Universal Robots PolyScope program: target_pose_tracking.urp

Program target_pose_tracking (createdIn=3.5.4.10845 lastSavedIn=3.5.4.10845 directory=/home/ur/ursim-current/programs installation=default robotSerialNumber=2014309999)
Calibrated DH parameters: a=[0, -0.612, -0.5723, 0, 0, 0]; d=[0.1273, 0, 0, 0.163941, 0.1157, 0.0922]; alpha=[1.570796, 0, 0, 1.570796, -1.570796, 0]; deltaTheta=[0, 0, 0, 0, 0, 0]
BeforeStart
  target_pose := Joint_6_name
  Popup Message (haltProgram=false message=Program has started from the beginning :D)
Robot Program (runOnlyOnce=false motionType=MoveJ speed=1.047198 acceleration=1.396263 useActiveTCP=false)
  Script: servoj(get_inverse_kin(target_pose))
  Script: sync()
Thread Thread_1 (runOnlyOnce=false trackProgramExecution=false)
  target_pose := Joint_6_name
  Loop Forever
    tmp := p[0,0,0,0,0,0]
    Script: tmp[0] = read_input_float_register(0)
    Script: tmp[1] = read_input_float_register(1)
    Script: tmp[2] = read_input_float_register(2)
    Script: tmp[3] = read_input_float_register(3)
    Script: tmp[4] = read_input_float_register(4)
    Script: tmp[5] = read_input_float_register(5)
    If tmp != p[0,0,0,0,0,0]
      target_pose := tmp
    Script: sync()
